Staubli VAL3: listAdd.pgx

program listAdd(string x_sEvent)
begin
  // add in the queue
  if sList!=""
    insert(sList[size(sList)])
  endIf
  sList[size(sList)-1]=x_sEvent
end
